FUNCTION_BLOCK E_Split5 (* Basic Function Block Type *)
  (* Standard: 61499-2 *)
  (* Version 0.0, 2011-02-28, Administrator, nxtControl GmbH, Template *)
  (* Compiler header: package fb.rt.pnp; *)
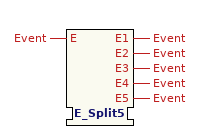
  EVENT_INPUT
    E; (* Normal Execution Request *)
  END_EVENT
  EVENT_OUTPUT
    E1; (* Execution Confirmation *)
    E2;
    E3;
    E4;
    E5;
  END_EVENT
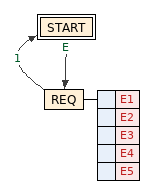
  EC_STATES
    START; (* Initial State *)
    REQ : -> E1, -> E2, -> E3, -> E4, -> E5; (* Normal execution *)
  END_STATES
  EC_TRANSITIONS
    START TO REQ := E;
    REQ TO START := 1;
  END_TRANSITIONS
  ALGORITHM INIT IN ST: (* Initialization algorithm *)
;
  END_ALGORITHM
  ALGORITHM REQ IN ST: (* Normally executed algorithm *)
;
  END_ALGORITHM
END_FUNCTION_BLOCK
